// TIA Portal V18 export
FUNCTION "ST10Cyl_interface71-80" : Void   // FC1027, LAD
{ S7_Optimized_Access := 'FALSE' }
VERSION : 0.1
// stored: AutoNumber false, IsIECCheckEnabled false, SetENOAutomatically false, UDAEnableTagReadback false
   VAR_INPUT
      AlwaysON : Bool;
      E_stop : Bool;
   END_VAR
   VAR_TEMP
      tTest : Bool;
   END_VAR
BEGIN

REGION Network 1 (SCL): Cylinder 71-80 IO Interface (SCL)
   (*
   //Cylinder71 IO    K-reserveTakeStopperCylinder1_1
   //Input
   "ST10Cylinder".Cy[71].In.WorkPositionSensor := "oK-reserveTakeStopperCylinder1_1";
   "ST10Cylinder".Cy[71].In.HomePositionSensor := NOT "oK-reserveTakeStopperCylinder1_1";
   //Output
   "oK-reserveTakeStopperCylinder1_1" := "ST10Cylinder".Cy[71].Out.GoWorkPosition;
   #tTest := "ST10Cylinder".Cy[71].Out.GoHomePosition;

   //Cylinder72 IO    K-reserveTakeStopperCylinder1_2
   //Input
   "ST10Cylinder".Cy[72].In.WorkPositionSensor := "oK-reserveTakeStopperCylinder1_2";
   "ST10Cylinder".Cy[72].In.HomePositionSensor := NOT "oK-reserveTakeStopperCylinder1_2";
   //Output
   "oK-reserveTakeStopperCylinder1_2" := "ST10Cylinder".Cy[72].Out.GoWorkPosition;
   #tTest := "ST10Cylinder".Cy[72].Out.GoHomePosition;

   //Cylinder73 IO  K-reserveTakeStopperCylinder2_1
   //Input
   "ST10Cylinder".Cy[73].In.WorkPositionSensor := "oK-reserveTakeStopperCylinder2_1";
   "ST10Cylinder".Cy[73].In.HomePositionSensor := NOT "oK-reserveTakeStopperCylinder2_1";
   //Output
   "oK-reserveTakeStopperCylinder2_1" := "ST10Cylinder".Cy[73].Out.GoWorkPosition;
   #tTest := "ST10Cylinder".Cy[73].Out.GoHomePosition;

   //Cylinder74 IO  K-reserveTakeStopperCylinder2_2
   //Input
   "ST10Cylinder".Cy[74].In.WorkPositionSensor := "oK-reserveTakeStopperCylinder2_2";
   "ST10Cylinder".Cy[74].In.HomePositionSensor := NOT "oK-reserveTakeStopperCylinder2_2";
   //Output
   "oK-reserveTakeStopperCylinder2_2" := "ST10Cylinder".Cy[74].Out.GoWorkPosition;
   #tTest := "ST10Cylinder".Cy[74].Out.GoHomePosition;

   //Cylinder75 IO  K-reserveTakeStopperCylinder3_1
   //Input
   "ST10Cylinder".Cy[75].In.WorkPositionSensor := "oK-reserveTakeStopperCylinder3_1";
   "ST10Cylinder".Cy[75].In.HomePositionSensor := NOT "oK-reserveTakeStopperCylinder3_1";
   //Output
   "oK-reserveTakeStopperCylinder3_1" := "ST10Cylinder".Cy[75].Out.GoWorkPosition;
   #tTest := "ST10Cylinder".Cy[75].Out.GoHomePosition;

   //Cylinder76 IO  K-reserveTakeStopperCylinder3_2
   //Input
   "ST10Cylinder".Cy[76].In.WorkPositionSensor := "oK-reserveTakeStopperCylinder3_2";
   "ST10Cylinder".Cy[76].In.HomePositionSensor := NOT "oK-reserveTakeStopperCylinder3_2";
   //Output
   "oK-reserveTakeStopperCylinder3_2" := "ST10Cylinder".Cy[76].Out.GoWorkPosition;
   #tTest := "ST10Cylinder".Cy[76].Out.GoHomePosition;

   *)
END_REGION

REGION Network 2: CY71 interface K-reserveTakeStopperCylinder1_1
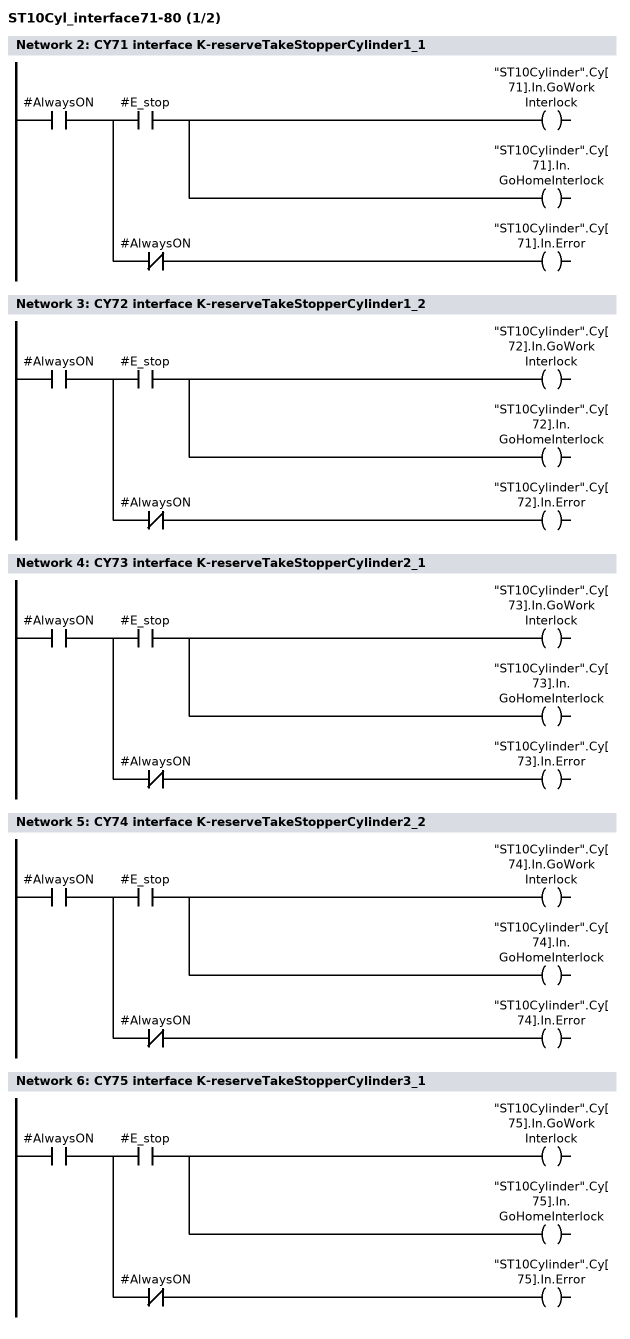
   RUNG wire#powerrail
      Contact( #AlwaysON )
      wire#w1
      Contact( #E_stop )
      wire#w2
      Coil( "ST10Cylinder".Cy[71].In.GoWorkInterlock )
   END_RUNG
   RUNG wire#w2
      Coil( "ST10Cylinder".Cy[71].In.GoHomeInterlock )
   END_RUNG
   RUNG wire#w1
      I_Contact( #AlwaysON )
      Coil( "ST10Cylinder".Cy[71].In.Error )
   END_RUNG
   // the same network as SCL:
   "ST10Cylinder".Cy[71].In.GoWorkInterlock := #AlwaysON AND #E_stop;
   "ST10Cylinder".Cy[71].In.GoHomeInterlock := #AlwaysON AND #E_stop;
   "ST10Cylinder".Cy[71].In.Error := #AlwaysON AND NOT #AlwaysON;
END_REGION

REGION Network 3: CY72 interface K-reserveTakeStopperCylinder1_2
   RUNG wire#powerrail
      Contact( #AlwaysON )
      wire#w1
      Contact( #E_stop )
      wire#w2
      Coil( "ST10Cylinder".Cy[72].In.GoWorkInterlock )
   END_RUNG
   RUNG wire#w2
      Coil( "ST10Cylinder".Cy[72].In.GoHomeInterlock )
   END_RUNG
   RUNG wire#w1
      I_Contact( #AlwaysON )
      Coil( "ST10Cylinder".Cy[72].In.Error )
   END_RUNG
   // the same network as SCL:
   "ST10Cylinder".Cy[72].In.GoWorkInterlock := #AlwaysON AND #E_stop;
   "ST10Cylinder".Cy[72].In.GoHomeInterlock := #AlwaysON AND #E_stop;
   "ST10Cylinder".Cy[72].In.Error := #AlwaysON AND NOT #AlwaysON;
END_REGION

REGION Network 4: CY73 interface K-reserveTakeStopperCylinder2_1
   RUNG wire#powerrail
      Contact( #AlwaysON )
      wire#w1
      Contact( #E_stop )
      wire#w2
      Coil( "ST10Cylinder".Cy[73].In.GoWorkInterlock )
   END_RUNG
   RUNG wire#w2
      Coil( "ST10Cylinder".Cy[73].In.GoHomeInterlock )
   END_RUNG
   RUNG wire#w1
      I_Contact( #AlwaysON )
      Coil( "ST10Cylinder".Cy[73].In.Error )
   END_RUNG
   // the same network as SCL:
   "ST10Cylinder".Cy[73].In.GoWorkInterlock := #AlwaysON AND #E_stop;
   "ST10Cylinder".Cy[73].In.GoHomeInterlock := #AlwaysON AND #E_stop;
   "ST10Cylinder".Cy[73].In.Error := #AlwaysON AND NOT #AlwaysON;
END_REGION

REGION Network 5: CY74 interface K-reserveTakeStopperCylinder2_2
   RUNG wire#powerrail
      Contact( #AlwaysON )
      wire#w1
      Contact( #E_stop )
      wire#w2
      Coil( "ST10Cylinder".Cy[74].In.GoWorkInterlock )
   END_RUNG
   RUNG wire#w2
      Coil( "ST10Cylinder".Cy[74].In.GoHomeInterlock )
   END_RUNG
   RUNG wire#w1
      I_Contact( #AlwaysON )
      Coil( "ST10Cylinder".Cy[74].In.Error )
   END_RUNG
   // the same network as SCL:
   "ST10Cylinder".Cy[74].In.GoWorkInterlock := #AlwaysON AND #E_stop;
   "ST10Cylinder".Cy[74].In.GoHomeInterlock := #AlwaysON AND #E_stop;
   "ST10Cylinder".Cy[74].In.Error := #AlwaysON AND NOT #AlwaysON;
END_REGION

REGION Network 6: CY75 interface K-reserveTakeStopperCylinder3_1
   RUNG wire#powerrail
      Contact( #AlwaysON )
      wire#w1
      Contact( #E_stop )
      wire#w2
      Coil( "ST10Cylinder".Cy[75].In.GoWorkInterlock )
   END_RUNG
   RUNG wire#w2
      Coil( "ST10Cylinder".Cy[75].In.GoHomeInterlock )
   END_RUNG
   RUNG wire#w1
      I_Contact( #AlwaysON )
      Coil( "ST10Cylinder".Cy[75].In.Error )
   END_RUNG
   // the same network as SCL:
   "ST10Cylinder".Cy[75].In.GoWorkInterlock := #AlwaysON AND #E_stop;
   "ST10Cylinder".Cy[75].In.GoHomeInterlock := #AlwaysON AND #E_stop;
   "ST10Cylinder".Cy[75].In.Error := #AlwaysON AND NOT #AlwaysON;
END_REGION

REGION Network 7: CY76 interface K-reserveTakeStopperCylinder3_2
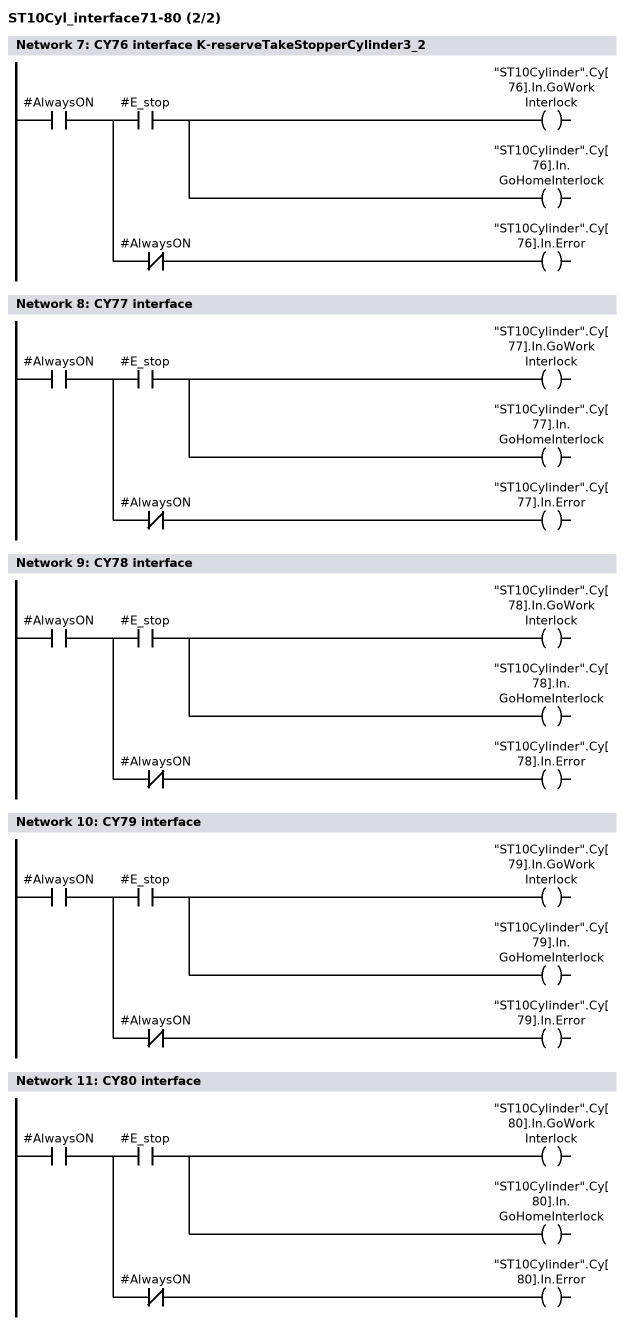
   RUNG wire#powerrail
      Contact( #AlwaysON )
      wire#w1
      Contact( #E_stop )
      wire#w2
      Coil( "ST10Cylinder".Cy[76].In.GoWorkInterlock )
   END_RUNG
   RUNG wire#w2
      Coil( "ST10Cylinder".Cy[76].In.GoHomeInterlock )
   END_RUNG
   RUNG wire#w1
      I_Contact( #AlwaysON )
      Coil( "ST10Cylinder".Cy[76].In.Error )
   END_RUNG
   // the same network as SCL:
   "ST10Cylinder".Cy[76].In.GoWorkInterlock := #AlwaysON AND #E_stop;
   "ST10Cylinder".Cy[76].In.GoHomeInterlock := #AlwaysON AND #E_stop;
   "ST10Cylinder".Cy[76].In.Error := #AlwaysON AND NOT #AlwaysON;
END_REGION

REGION Network 8: CY77 interface
   RUNG wire#powerrail
      Contact( #AlwaysON )
      wire#w1
      Contact( #E_stop )
      wire#w2
      Coil( "ST10Cylinder".Cy[77].In.GoWorkInterlock )
   END_RUNG
   RUNG wire#w2
      Coil( "ST10Cylinder".Cy[77].In.GoHomeInterlock )
   END_RUNG
   RUNG wire#w1
      I_Contact( #AlwaysON )
      Coil( "ST10Cylinder".Cy[77].In.Error )
   END_RUNG
   // the same network as SCL:
   "ST10Cylinder".Cy[77].In.GoWorkInterlock := #AlwaysON AND #E_stop;
   "ST10Cylinder".Cy[77].In.GoHomeInterlock := #AlwaysON AND #E_stop;
   "ST10Cylinder".Cy[77].In.Error := #AlwaysON AND NOT #AlwaysON;
END_REGION

REGION Network 9: CY78 interface
   RUNG wire#powerrail
      Contact( #AlwaysON )
      wire#w1
      Contact( #E_stop )
      wire#w2
      Coil( "ST10Cylinder".Cy[78].In.GoWorkInterlock )
   END_RUNG
   RUNG wire#w2
      Coil( "ST10Cylinder".Cy[78].In.GoHomeInterlock )
   END_RUNG
   RUNG wire#w1
      I_Contact( #AlwaysON )
      Coil( "ST10Cylinder".Cy[78].In.Error )
   END_RUNG
   // the same network as SCL:
   "ST10Cylinder".Cy[78].In.GoWorkInterlock := #AlwaysON AND #E_stop;
   "ST10Cylinder".Cy[78].In.GoHomeInterlock := #AlwaysON AND #E_stop;
   "ST10Cylinder".Cy[78].In.Error := #AlwaysON AND NOT #AlwaysON;
END_REGION

REGION Network 10: CY79 interface
   RUNG wire#powerrail
      Contact( #AlwaysON )
      wire#w1
      Contact( #E_stop )
      wire#w2
      Coil( "ST10Cylinder".Cy[79].In.GoWorkInterlock )
   END_RUNG
   RUNG wire#w2
      Coil( "ST10Cylinder".Cy[79].In.GoHomeInterlock )
   END_RUNG
   RUNG wire#w1
      I_Contact( #AlwaysON )
      Coil( "ST10Cylinder".Cy[79].In.Error )
   END_RUNG
   // the same network as SCL:
   "ST10Cylinder".Cy[79].In.GoWorkInterlock := #AlwaysON AND #E_stop;
   "ST10Cylinder".Cy[79].In.GoHomeInterlock := #AlwaysON AND #E_stop;
   "ST10Cylinder".Cy[79].In.Error := #AlwaysON AND NOT #AlwaysON;
END_REGION

REGION Network 11: CY80 interface
   RUNG wire#powerrail
      Contact( #AlwaysON )
      wire#w1
      Contact( #E_stop )
      wire#w2
      Coil( "ST10Cylinder".Cy[80].In.GoWorkInterlock )
   END_RUNG
   RUNG wire#w2
      Coil( "ST10Cylinder".Cy[80].In.GoHomeInterlock )
   END_RUNG
   RUNG wire#w1
      I_Contact( #AlwaysON )
      Coil( "ST10Cylinder".Cy[80].In.Error )
   END_RUNG
   // the same network as SCL:
   "ST10Cylinder".Cy[80].In.GoWorkInterlock := #AlwaysON AND #E_stop;
   "ST10Cylinder".Cy[80].In.GoHomeInterlock := #AlwaysON AND #E_stop;
   "ST10Cylinder".Cy[80].In.Error := #AlwaysON AND NOT #AlwaysON;
END_REGION
END_FUNCTION
